% RSLogix 500 project MODBUS_PULSOS_PID_BAK472.RSS, saved by version 7.30.00.17 %
PROJECT "UNTITLED"    % processor: Bul.1763 MicroLogix 1100 Series B %

PROGRAM FILES
  LAD 2 "PRINCIPAL"  4 rungs
  LAD 3 "MODBUS"  5 rungs
  LAD 4 "COMANDOS"  8 rungs
  LAD 5 "HSC_SUB"  5 rungs
  LAD 6 "CONTROL"  10 rungs

DATA FILES
  O0 OUTPUT  4 elements
  I1 INPUT  6 elements
  S2 STATUS  66 elements
  B3 BINARY  1 elements
  T4 TIMER  1 elements
  C5 COUNTER  1 elements
  R6 CONTROL  1 elements
  N7 INTEGER  15 elements
  F8 FLOAT  10 elements
  PD9   1 elements
  MG11   5 elements

LADDER 2 "PRINCIPAL"
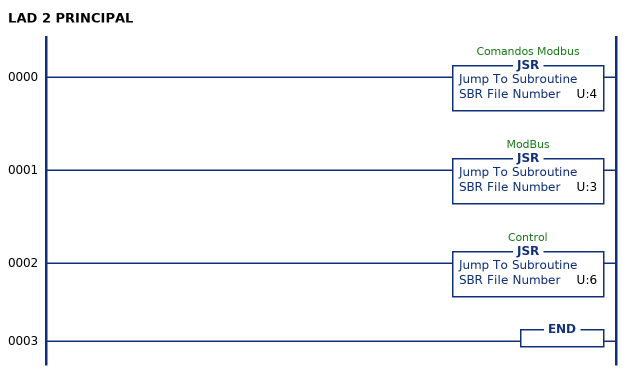
% Rung: 0 %
SOR JSR U:4 EOR
%   U:4  "Comandos Modbus" %
% Rung: 1 %
SOR JSR U:3 EOR
%   U:3  "ModBus" %
% Rung: 2 %
SOR JSR U:6 EOR
%   U:6  "Control" %
% Rung: 3 %
SOR END EOR

LADDER 3 "MODBUS"
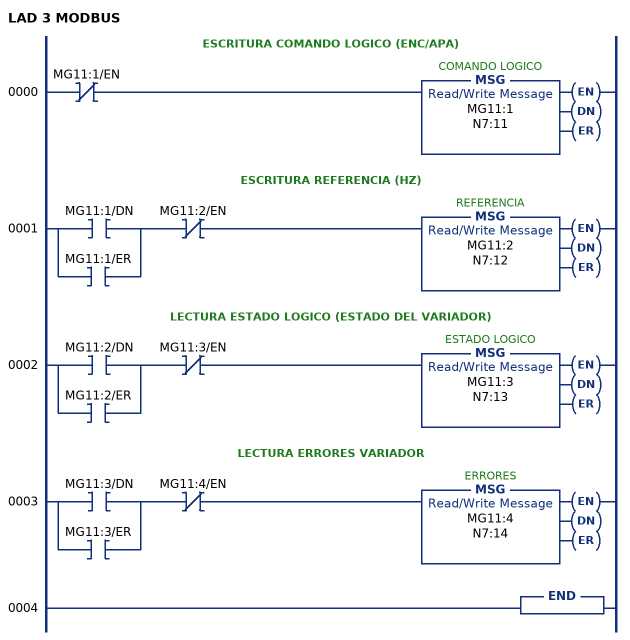
% Rung: 0 %
% TITLE: ESCRITURA COMANDO LOGICO (ENC/APA) %
SOR XIO MG11:1/EN MSG MG11:1 N7:11 EOR
%   MSG set-up: 06 Write Single Register (4xxxxx) | 2 | 1 | 8193 | N7:11 | 0 | 100 | 0 | CLIENT | 0 | 0 | ? %
%   MG11:1  "COMANDO LOGICO" %
%   N7:11  "COMANDO LOGICO" %
% Rung: 1 %
% TITLE: ESCRITURA REFERENCIA (HZ) %
SOR BST XIC MG11:1/DN NXB XIC MG11:1/ER BND XIO MG11:2/EN MSG MG11:2 N7:12 EOR
%   MSG set-up: 06 Write Single Register (4xxxxx) | 2 | 1 | 8194 | N7:12 | 0 | 100 | 0 | CLIENT | 0 | 0 | ? %
%   MG11:2  "REFERENCIA" %
%   N7:12  "ESFUERZO" %
% Rung: 2 %
% TITLE: LECTURA ESTADO LOGICO (ESTADO DEL VARIADOR) %
SOR BST XIC MG11:2/DN NXB XIC MG11:2/ER BND XIO MG11:3/EN MSG MG11:3 N7:13 EOR
%   MSG set-up: 03 Read Holding Registers (4xxxxx) | 2 | 1 | 8449 | N7:13 | 0 | 100 | 0 | CLIENT | 0 | 0 | ? %
%   MG11:3  "ESTADO LOGICO" %
%   N7:13  "ESTADO LOGICO" %
% Rung: 3 %
% TITLE: LECTURA ERRORES VARIADOR %
SOR BST XIC MG11:3/DN NXB XIC MG11:3/ER BND XIO MG11:4/EN MSG MG11:4 N7:14 EOR
%   MSG set-up: 03 Read Holding Registers (4xxxxx) | 2 | 1 | 8450 | N7:14 | 0 | 100 | 0 | CLIENT | 0 | 0 | ? %
%   MG11:4  "ERRORES" %
%   N7:14  "ERRORES" %
% Rung: 4 %
SOR END EOR

LADDER 4 "COMANDOS"
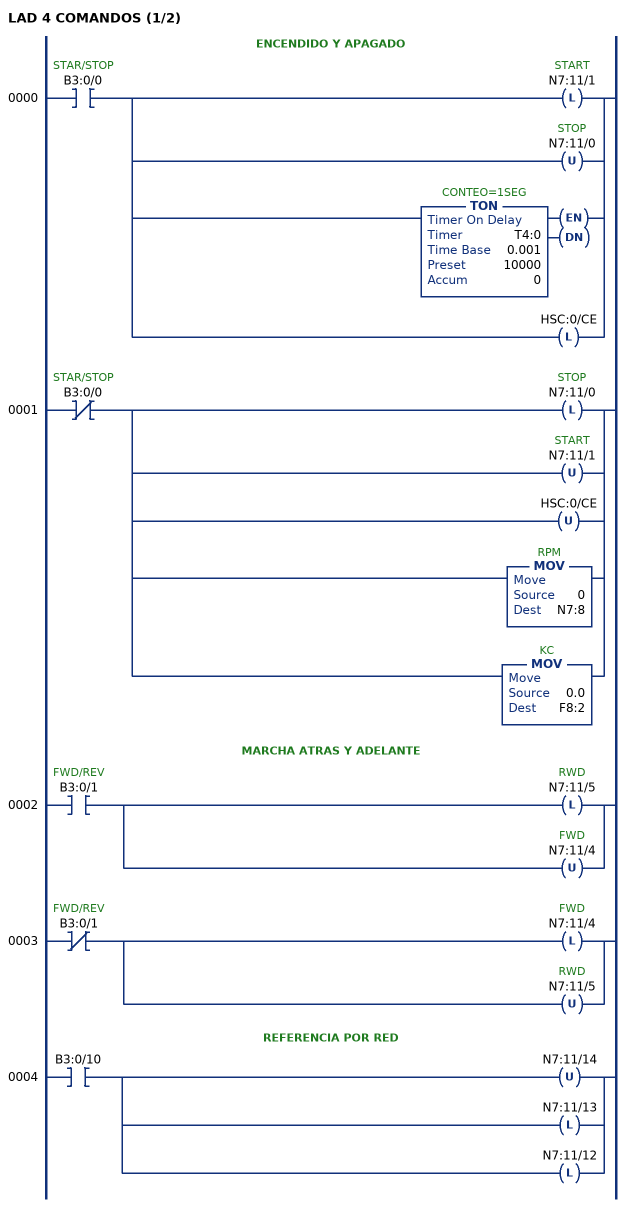
% Rung: 0 %
% TITLE: ENCENDIDO Y APAGADO %
SOR XIC B3:0/0 BST OTL N7:11/1 NXB OTU N7:11/0 NXB TON T4:0 0.001 10000 0 NXB OTL HSC:0/CE BND EOR
%   B3:0/0  "STAR/STOP" %
%   N7:11/1  "START" %
%   N7:11/0  "STOP" %
%   T4:0  "CONTEO=1SEG" %
% Rung: 1 %
SOR XIO B3:0/0 BST OTL N7:11/0 NXB OTU N7:11/1 NXB OTU HSC:0/CE NXB MOV 0 N7:8 NXB MOV 0.0 F8:2 BND EOR
%   B3:0/0  "STAR/STOP" %
%   N7:11/0  "STOP" %
%   N7:11/1  "START" %
%   N7:8  "RPM" %
%   F8:2  "KC" %
% Rung: 2 %
% TITLE: MARCHA ATRAS Y ADELANTE %
SOR XIC B3:0/1 BST OTL N7:11/5 NXB OTU N7:11/4 BND EOR
%   B3:0/1  "FWD/REV" %
%   N7:11/5  "RWD" %
%   N7:11/4  "FWD" %
% Rung: 3 %
SOR XIO B3:0/1 BST OTL N7:11/4 NXB OTU N7:11/5 BND EOR
%   B3:0/1  "FWD/REV" %
%   N7:11/4  "FWD" %
%   N7:11/5  "RWD" %
% Rung: 4 %
% TITLE: REFERENCIA POR RED %
SOR XIC B3:0/10 BST OTU N7:11/14 NXB OTL N7:11/13 NXB OTL N7:11/12 BND EOR

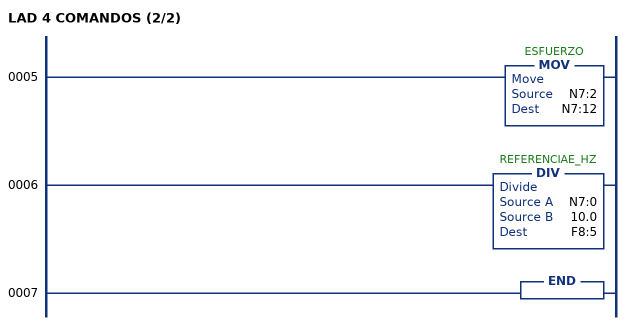
% Rung: 5 %
SOR MOV N7:2 N7:12 EOR
%   N7:2  "SALIDA-PID-%" %
%   N7:12  "ESFUERZO" %
% Rung: 6 %
SOR DIV N7:0 10.0 F8:5 EOR
%   N7:0  "SP-FRECUENCIA" %
%   F8:5  REFERENCIAE_HZ %
% Rung: 7 %
SOR END EOR

LADDER 5 "HSC_SUB"
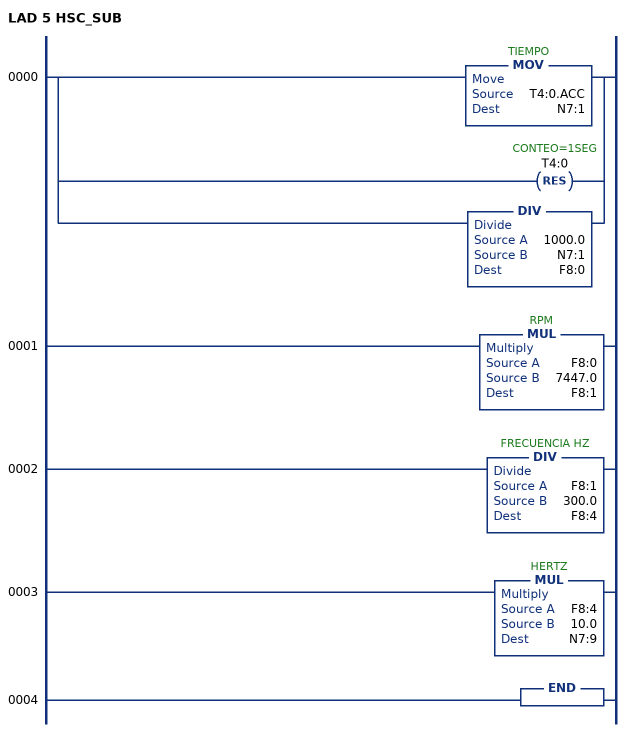
% Rung: 0 %
SOR BST MOV T4:0.ACC N7:1 NXB RES T4:0 NXB DIV 1000.0 N7:1 F8:0 BND EOR
%   T4:0  "CONTEO=1SEG" %
%   N7:1  "TIEMPO" %
% Rung: 1 %
SOR MUL F8:0 7447.0 F8:1 EOR
%   F8:1  "RPM" %
% Rung: 2 %
SOR DIV F8:1 300.0 F8:4 EOR
%   F8:1  "RPM" %
%   F8:4  "FRECUENCIA HZ" %
% Rung: 3 %
SOR MUL F8:4 10.0 N7:9 EOR
%   F8:4  "FRECUENCIA HZ" %
%   N7:9  "HERTZ" %
% Rung: 4 %
SOR END EOR

LADDER 6 "CONTROL"
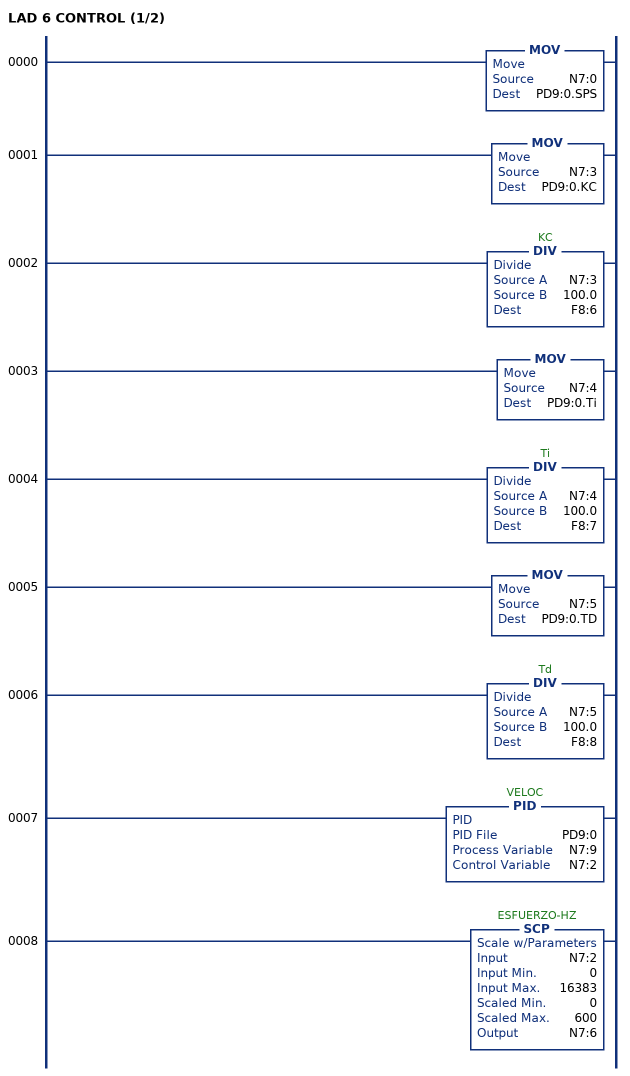
% Rung: 0 %
SOR MOV N7:0 PD9:0.SPS EOR
%   N7:0  "SP-FRECUENCIA" %
% Rung: 1 %
SOR MOV N7:3 PD9:0.KC EOR
%   N7:3  "KP" %
% Rung: 2 %
SOR DIV N7:3 100.0 F8:6 EOR
%   N7:3  "KP" %
%   F8:6  "KC" %
% Rung: 3 %
SOR MOV N7:4 PD9:0.Ti EOR
%   N7:4  "TI" %
% Rung: 4 %
SOR DIV N7:4 100.0 F8:7 EOR
%   N7:4  "TI" %
%   F8:7  "Ti" %
% Rung: 5 %
SOR MOV N7:5 PD9:0.TD EOR
%   N7:5  "TD" %
% Rung: 6 %
SOR DIV N7:5 100.0 F8:8 EOR
%   N7:5  "TD" %
%   F8:8  "Td" %
% Rung: 7 %
SOR PID PD9:0 N7:9 N7:2 EOR
%   PD9:0  VELOC %
%   N7:9  "HERTZ" %
%   N7:2  "SALIDA-PID-%" %
% Rung: 8 %
SOR SCP N7:2 0 16383 0 600 N7:6 EOR
%   N7:2  "SALIDA-PID-%" %
%   N7:6  "ESFUERZO-HZ" %

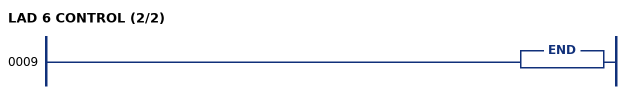
% Rung: 9 %
SOR END EOR

OTHER DOCUMENTED ADDRESSES
  B3:0/2  "DIST. ON"
  I:1.1  PRESION_ENTRA_TX_HW
  O:0.0/0  "DISTURBIO"
  PFILE:5  "HSC"
  U:5  "HSC"

COMMENTS NOT ATTACHED TO A CURRENT RUNG
  N12:0/5: FWD
  N12:0/2: JOG
  MG11:0: ESCRITURA COMANDO LOGICO (ENC/APA)
  MG11:1: REFERENCIA
  MG11:2: DATOS DE ESTADO LOGICO
  MG11:3: FRECUENCIA
  MG11:4: FALLAS

REVISION NOTES
  0: Cambiado tiempo

DATA TABLE (non-zero values as saved)
DATA B3
% B3:0 % 0X0400
DATA T4
% .PRE .ACC %
% T4:0 % 10000 0
DATA N7
% N7:0 % 0 696 445 0 0 0 16 0 0 357
% N7:10 % 0 12322 655 1795 0
DATA F8
% F8:0 % 1.436782 10699.71 0 7 35.66571
% F8:5 % 50 0 0 0 0
